// SIMATIC S7-200 SMART project (STEP 7-Micro/WIN SMART), CPU ST60

SYMBOL_TABLE 表格 1
RamZ             I0.0     // 压头零点
LeftStepPosLimit I0.1     // 左步进机构正限位
LeftStepNegaLimt I0.2     // 左步进机构负限位
RightStepPosLimit I0.3     // 右步进机构正限位
RightStepNegaLimt I0.4     // 右步进机构负限位
AirDownLimit     I0.5     // 气囊下限位
AirUpLimit       I0.6     // 气囊上限位
EMBotton         I0.7     // 急停
JOG1             I1.0     // JOG-
JOG2             I1.1     // JOG+
ResetBotton      I1.2     // 复位按钮
StartBotton      I1.3     // 循环启动
ManualBotton     I1.4     // 手动
AutoBotton       I1.5     // 自动
InderRunDone     I1.7     // 压头运行到位完成
Step1UpLimit     I2.0     // 步进机构气缸1上限位
Step1DownLimit   I2.1     // 步进机构气缸1下限位
Step2UpLimit     I2.2     // 步进机构气缸2上限位
Step2DownLimit   I2.3     // 步进机构气缸2下限位
LeftTopDownLimit I2.4     // 左顶尖气缸下限位
RightTopDownLimit I2.5     // 右顶尖气缸下限位
PipaBackLimit    I2.6     // 琵琶孔退回到位1
Ram1_Ready       I2.7     // 压头1伺服准备
Ram1_Alarm       I3.0     // 压头1驱动报警
Rot_Alarm        I3.1     // 旋转电机报警
Step_Alarm       I3.2     // 步进电机报警
PipaBackLimit2   I3.3     // 琵琶孔退回到位2
Ram2_Ready       I3.4     // 压头2伺服准备
Ram2_Alarm       I3.5     // 压头2驱动报警
Step_Send        I3.6     // 步进机构可送料信号
Step_First       I3.7     // 步进机构首端有料
Step_Middle      I4.0     // 校直机有料
Step_Last        I4.1     // 步进机构末端有料
LeftClamClose    I4.2     // 左夹爪气缸夹紧到位
RightClamClose   I4.3     // 右夹爪气缸夹紧到位
Press_Abnormal   I12.0    // 气压异常
FloatSup1BackLimit I12.1    // 浮动支撑1退回到位
FloatSup2BackLimit I12.2    // 浮动支撑2退回到位
FloatSup3BackLimit I12.3    // 浮动支撑3退回到位
FloatSup4BackLimit I12.4    // 浮动支撑4退回到位
FloatSup1FrontLimit I12.5    // 浮动支撑1前进到位
FloatSup2FrontLimit I12.6    // 浮动支撑2前进到位
FloatSup3FrontLimit I12.7    // 浮动支撑3前进到位
FloatSup4FrontLimit I16.0    // 浮动支撑4前进到位
YT5_BackLimit    I16.1    // 压头5缩回到位
YT4_BackLimit    I16.2    // 压头4缩回到位
YT3_BackLimit    I16.3    // 压头3缩回到位
YT2_BackLimit    I16.4    // 压头2缩回到位
YT1_BackLimit    I16.5    // 压头1缩回到位
LeftTopFloatLimit I16.6    // 左顶尖前进到位
LeftTopBackLimit I16.7    // 左顶尖退回到位
RightTopFloatLimit I17.0    // 右顶尖前进到位
RightTopBackLimit I17.1    // 右顶尖退回到位
找平到位             I17.3
步进后退             M11.0
步进前进             M11.2
主轴抬起             M11.4
主轴下压             M11.6
找平升              M12.0
支撑1进             M12.2
支撑2进             M12.3
支撑3进             M12.4
支撑4进             M12.5
一次抬起             M12.7
一次下压             M12.6
结束计时             M14.1
下压轴停止信号          M13.0
RamPULS          Q0.0     // 压头脉冲
StepPULS         Q0.1     // 左步进脉冲
RamSIGN          Q0.2     // 压头方向：高电位时压头下移，位移为正
RotaPULS         Q0.3     // 右步进电机脉冲
StartLamp        Q0.4     // 循环启动按钮灯
ServStart        Q0.5     // 启动
Ram_Rest         Q0.6     // 压头报警复位
Step_Sign        Q0.7     // 左步进机构方向
RotoSIGN         Q1.0     // 右旋转电机方向
YT1              Q1.2     // 1号压头气缸
YT2              Q1.3     // 2号压头气缸
YT3              Q1.4     // 3号压头气缸
YT4              Q1.5     // 4号压头气缸
YT5              Q1.6     // 5号压头气缸
Pipahole_Measure Q1.7     // 琵琶孔测量气缸
FloatSupport1    Q2.0     // 浮动支撑1缩回
FloatSupport2    Q2.1     // 浮动支撑2缩回
FloatSupport3    Q2.2     // 浮动支撑3缩回
FloatSupport4    Q2.3     // 浮动支撑4缩回
TopClamp         Q2.4     // 顶尖气缸夹紧
TopRelease       Q2.5     // 顶尖气缸松开
TopForward       Q2.6     // 顶尖气缸前进
Topback          Q2.7     // 顶尖气缸缩回
InderAirbagUp    Q8.0     // 压头气囊升起
InderAirbagDown  Q8.1     // 压头气囊落下
StepDown2        Q8.2     // 步进机构1落下
StepUp2          Q8.3     // 步进机构1升起
TopUp            Q8.4     // 顶尖气缸升起
TopDown          Q8.5     // 顶尖气缸落下
StepLast         Q8.6     // 步进机构末端可取料信号
FM               Q9.0     // 蜂鸣器
GREEN            Q9.1     // 绿灯
YELLOW           Q9.2     // 黄灯
RED              Q9.3     // 红灯
HG               Q9.4     // 加工合格
BHG              Q9.5     // 加工不合格
平升               Q12.0
左步进错误            VB300
右步进错误            VB304
下压轴错误            VB308
左步进速度            VD400
右步进速度            VD404
下压轴速度            VD408
左步进pos           VD412
右步进pos           VD416
下压轴pos           VD420
END_SYMBOL_TABLE

SYMBOL_TABLE 表格 2
HSC0_FREQ_PERIOD SMB196   // HSC0 频率测量周期: 0=1s 1=100ms 2=10ms
HSC0_TYPE        SMB195   // HSC0 类型: 0=计数 1=频率
HSC1_FREQ_PERIOD SMB198   // HSC1 频率测量周期: 0=1s 1=100ms 2=10ms
HSC1_TYPE        SMB197   // HSC1 类型: 0=计数 1=频率
HSC2_FREQ_PERIOD SMB200   // HSC2 频率测量周期: 0=1s 1=100ms 2=10ms
HSC2_TYPE        SMB199   // HSC2 类型: 0=计数 1=频率
HSC3_FREQ_PERIOD SMB202   // HSC3 频率测量周期: 0=1s 1=100ms 2=10ms
HSC3_TYPE        SMB201   // HSC3 类型: 0=计数 1=频率
HSC4_FREQ_PERIOD SMB204   // HSC4 频率测量周期: 0=1s 1=100ms 2=10ms
HSC4_TYPE        SMB203   // HSC4 类型: 0=计数 1=频率
HSC5_FREQ_PERIOD SMB206   // HSC5 频率测量周期: 0=1s 1=100ms 2=10ms
HSC5_TYPE        SMB205   // HSC5 类型: 0=计数 1=频率
PLS3_Abort_AE    SM580.4  // 由于添加错误终止 PTO2 包络：0 = 未终止；1 = 终止
PLS3_Ctrl        SMB581   // 监视和控制 Q0.2 的 PTO3（脉冲串输出）和 PWM3（脉冲宽度调制）
PLS3_Cycle       SMW582   // PWM3 周期值（2 到 65,535 个单位时基）；PTO3 频率值（1 到 65,535 Hz）
PLS3_Cycle_Update SM581.0  // PTO3/PWM3 更新周期或频率值：0 = 不更新；1 = 写入新周期/频率
PLS3_Disable_UC  SM580.5  // PTO3 用户在 PTO 包络运行过程中手动将其禁用 ：0 = 未禁用；1 = 手动禁用
PLS3_Enable      SM581.7  // PTO3/PWM3 使能：0 = 禁用；1 = 启用。
PLS3_Idle        SM580.7  // PTO3 空闲：0 = PTO 正在执行；1 = PTO 空闲。
PLS3_Ovr         SM580.6  // PTO3 管道上溢/下溢，管道为满时装载管道或传送空管道时：0 = 无溢出，1 = 管道上溢/下溢
PLS3_Select      SM581.6  // PTO3/PWM3 模式选择：0 = PWM；1 = PTO。
PTO3_Operation   SM581.5  // PTO3 选择单段/多段操作： 0 = 单段操作；1 = 多段操作
PTO3_PC          SMD586   // PTO3 脉冲计数值（1 到 2^32 - 1）
PTO3_PC_Update   SM581.2  // PTO3 更新脉冲计数值：0 = 不更新；1 = 写入新脉冲计数
PTO3_Profile_Offset SMW592   // PTO3 包络表的起始位置（从 V0 开始字节偏移）
PTO3_Seg_Num     SMB590   // 当前执行的 PTO3 包络的段数
PTO3_Status      SMB580   // PTO3 状态
PWM3_PW          SMW584   // PWM3 脉冲宽度值（0 到 65,535 个单位时基）
PWM3_PW_Update   SM581.1  // PWM3 更新脉冲宽度值：0 = 不更新；1 = 写入新脉冲宽度
PWM3_TimeBase    SM581.3  // PWM3 时基：0 = 1μs/刻度，1 = 1ms/刻度
END_SYMBOL_TABLE

SYMBOL_TABLE 表格 3
步进上料自锁           M0.0
夹正PC             M0.1
夹升PC             M0.2
夹反PC             M0.3
夹退PC             M0.4
夹停PC             M0.5
夹进PC             M0.6
夹紧PC             M0.7
夹降PC             M1.0
夹松PC             M1.1
步回零              M1.2
步最后PC            M1.3
步回零PC            M1.4
步最前PC            M1.5
步后PC             M1.6
步停PC             M1.7
步前PC             M2.0
步升PC             M2.1
步降PC             M2.2
axis0_dir        M2.3
压1进PC            M2.4
压1退PC            M2.5
压2进PC            M2.6
压2退PC            M2.7
压3进PC            M3.0
压3退PC            M3.1
压4进PC            M3.2
压4退PC            M3.3
压5进PC            M3.4
压5退PC            M3.5
压升PC             M3.6
压降PC             M3.7
压停PC             M4.0
压回零PC            M4.1
充气PC             M4.2
停充PC             M4.3
放气PC             M4.4
平升PC             M4.5
平停PC             M4.6
平降PC             M4.7
撑1进PC            M5.0
撑1停PC            M5.1
撑1退PC            M5.2
撑2进PC            M5.3
撑2停PC            M5.4
撑2退PC            M5.5
撑3进PC            M5.6
撑3停PC            M5.7
撑3退PC            M6.0
撑4进PC            M6.1
撑4停PC            M6.2
撑4退PC            M6.3
夹爪复位             M6.4
夹爪准备             M6.5
进出料              M6.6
压real            M6.7
有料未出             M7.0
机械INIT           M7.1
init_isrun       M7.2
axis1_dir        M7.3
axis0_动作         M7.4
axis1_动作         M7.5
急停               M7.6
压回零重设done        M7.7
左步进done          M8.0
右步进done          M8.1
下压轴done          M8.2
左步进dir           M8.3
右步进dir           M8.4
下压轴dir           M8.5
压回零done          M8.6
左步回零done         M8.7
右步回零done         M9.0
NG               M9.1
test             M9.2     // OK
OK               M9.3
找平ok             M9.4
备压PC             M9.5
传感器有料            M9.7
出料后有料            M10.0
下压isrun          M10.1
PLC_EN           M10.2
（先出）请求上料PC       M10.3
步进isrun          M10.4
夹爪isrun          M10.5
（不出）请求上料pc       M10.6
心跳               M30.0
下料信号             M30.1
下压量              MD20
END_SYMBOL_TABLE

SYMBOL_TABLE 表格 4
input1           V701.0
input2           V701.1
input3           V701.2
input4           V701.3
input5           V701.4
input6           V701.5
input7           V701.6
input8           V701.7
input9           V702.0
input10          V702.1
input11          V702.2
input12          V702.3
input13          V702.4
input14          V702.5
input15          V702.6
input16          V702.7
inputrel1        VD703
inputrel2        VD707
inputrel3        VD711
inputrel4        VD715
inputrel5        VD719
inputrel6        VD723
inputrel7        VD727
inputrel8        VD731
output1          V801.0
output2          V801.1
output3          V801.2
output4          V801.3
output5          V801.4
output6          V801.5
output7          V801.6
output8          V801.7
output9          V802.0
output10         V802.1
output11         V802.2
output12         V802.3
output13         V802.4
output14         V802.5
output15         V802.6
output16         V802.7
outputrel1       VD803
outputrel2       VD807
outputrel3       VD811
outputrel4       VD815
outputrel5       VD819
outputrel6       VD823
outputrel7       VD827
outputrel8       VD831
END_SYMBOL_TABLE

ORGANIZATION_BLOCK MAIN:OB1
TITLE=程序注释
BEGIN
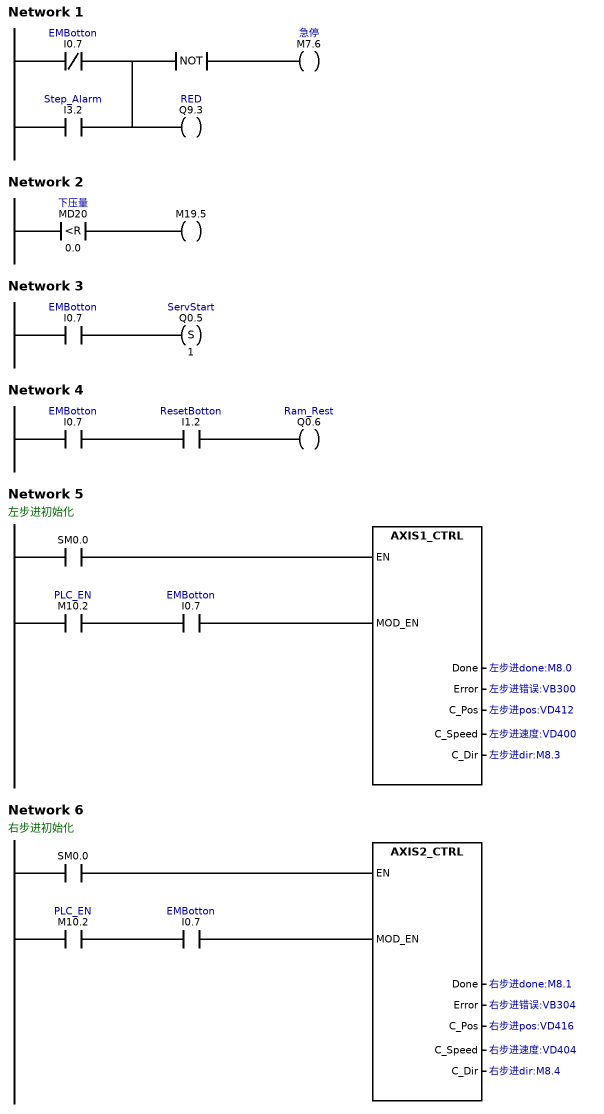
Network 1
LDN    EMBotton:I0.7
O      Step_Alarm:I3.2
LPS
NOT
=      急停:M7.6
LPP
=      RED:Q9.3
Network 2
LDR<   下压量:MD20, 0.0
=      M19.5
Network 3
LD     EMBotton:I0.7
S      ServStart:Q0.5, 1
Network 4
LD     EMBotton:I0.7
A      ResetBotton:I1.2
=      Ram_Rest:Q0.6
Network 5
// 左步进初始化
LD     SM0.0
=      L60.0
LD     PLC_EN:M10.2
A      EMBotton:I0.7
=      L63.7
LD     L60.0
CALL   AXIS1_CTRL:SBR12, L63.7, 左步进done:M8.0, 左步进错误:VB300, 左步进pos:VD412, 左步进速度:VD400, 左步进dir:M8.3
Network 6
// 右步进初始化
LD     SM0.0
=      L60.0
LD     PLC_EN:M10.2
A      EMBotton:I0.7
=      L63.7
LD     L60.0
CALL   AXIS2_CTRL:SBR23, L63.7, 右步进done:M8.1, 右步进错误:VB304, 右步进pos:VD416, 右步进速度:VD404, 右步进dir:M8.4
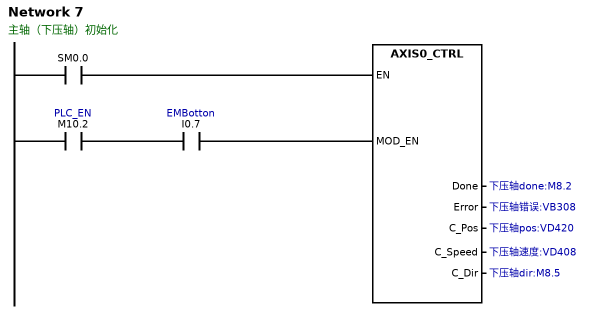
Network 7
// 主轴（下压轴）初始化
LD     SM0.0
=      L60.0
LD     PLC_EN:M10.2
A      EMBotton:I0.7
=      L63.7
LD     L60.0
CALL   AXIS0_CTRL:SBR4, L63.7, 下压轴done:M8.2, 下压轴错误:VB308, 下压轴pos:VD420, 下压轴速度:VD408, 下压轴dir:M8.5
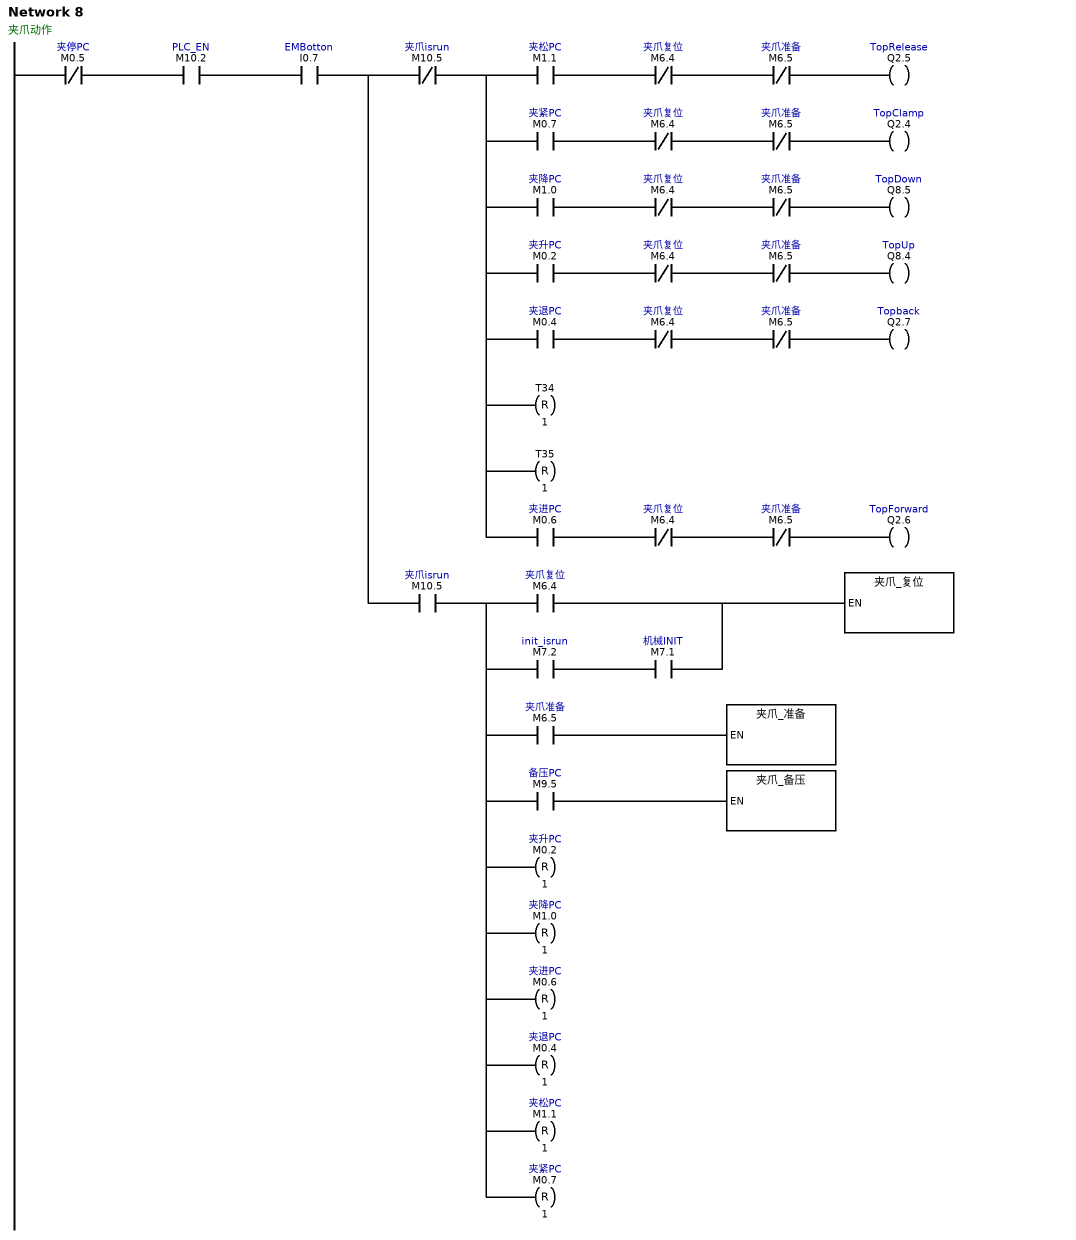
Network 8
// 夹爪动作
LDN    夹停PC:M0.5
A      PLC_EN:M10.2
A      EMBotton:I0.7
LPS
AN     夹爪isrun:M10.5
LPS
A      夹松PC:M1.1
AN     夹爪复位:M6.4
AN     夹爪准备:M6.5
=      TopRelease:Q2.5
LRD
A      夹紧PC:M0.7
AN     夹爪复位:M6.4
AN     夹爪准备:M6.5
=      TopClamp:Q2.4
LRD
A      夹降PC:M1.0
AN     夹爪复位:M6.4
AN     夹爪准备:M6.5
=      TopDown:Q8.5
LRD
A      夹升PC:M0.2
AN     夹爪复位:M6.4
AN     夹爪准备:M6.5
=      TopUp:Q8.4
LRD
A      夹退PC:M0.4
AN     夹爪复位:M6.4
AN     夹爪准备:M6.5
=      Topback:Q2.7
LRD
R      T34, 1
LRD
R      T35, 1
LPP
A      夹进PC:M0.6
AN     夹爪复位:M6.4
AN     夹爪准备:M6.5
=      TopForward:Q2.6
LPP
A      夹爪isrun:M10.5
LPS
LD     夹爪复位:M6.4
LD     init_isrun:M7.2
A      机械INIT:M7.1
OLD
ALD
CALL   夹爪_复位:SBR0
LPP
LPS
A      夹爪准备:M6.5
CALL   夹爪_准备:SBR1
LRD
A      备压PC:M9.5
CALL   夹爪_备压:SBR35
LRD
R      夹升PC:M0.2, 1
LRD
R      夹降PC:M1.0, 1
LRD
R      夹进PC:M0.6, 1
LRD
R      夹退PC:M0.4, 1
LRD
R      夹松PC:M1.1, 1
LPP
R      夹紧PC:M0.7, 1
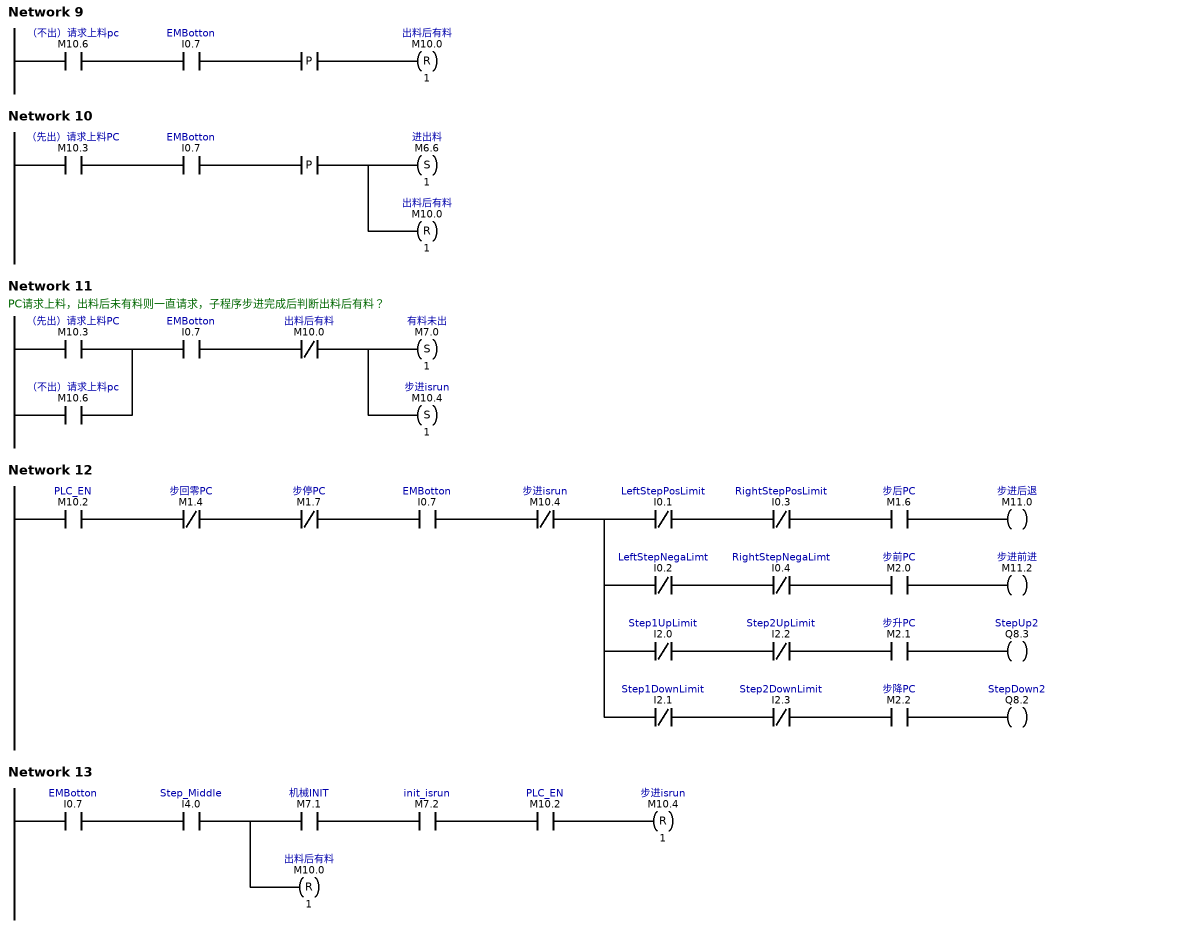
Network 9
LD     （不出）请求上料pc:M10.6
A      EMBotton:I0.7
EU
R      出料后有料:M10.0, 1
Network 10
LD     （先出）请求上料PC:M10.3
A      EMBotton:I0.7
EU
S      进出料:M6.6, 1
R      出料后有料:M10.0, 1
Network 11
// PC请求上料，出料后未有料则一直请求，子程序步进完成后判断出料后有料？
LD     （先出）请求上料PC:M10.3
O      （不出）请求上料pc:M10.6
A      EMBotton:I0.7
AN     出料后有料:M10.0
S      有料未出:M7.0, 1
S      步进isrun:M10.4, 1
Network 12
LD     PLC_EN:M10.2
AN     步回零PC:M1.4
AN     步停PC:M1.7
A      EMBotton:I0.7
AN     步进isrun:M10.4
LPS
AN     LeftStepPosLimit:I0.1
AN     RightStepPosLimit:I0.3
A      步后PC:M1.6
=      步进后退:M11.0
LRD
AN     LeftStepNegaLimt:I0.2
AN     RightStepNegaLimt:I0.4
A      步前PC:M2.0
=      步进前进:M11.2
LRD
AN     Step1UpLimit:I2.0
AN     Step2UpLimit:I2.2
A      步升PC:M2.1
=      StepUp2:Q8.3
LPP
AN     Step1DownLimit:I2.1
AN     Step2DownLimit:I2.3
A      步降PC:M2.2
=      StepDown2:Q8.2
Network 13
LD     EMBotton:I0.7
A      Step_Middle:I4.0
LPS
A      机械INIT:M7.1
A      init_isrun:M7.2
A      PLC_EN:M10.2
R      步进isrun:M10.4, 1
LPP
R      出料后有料:M10.0, 1
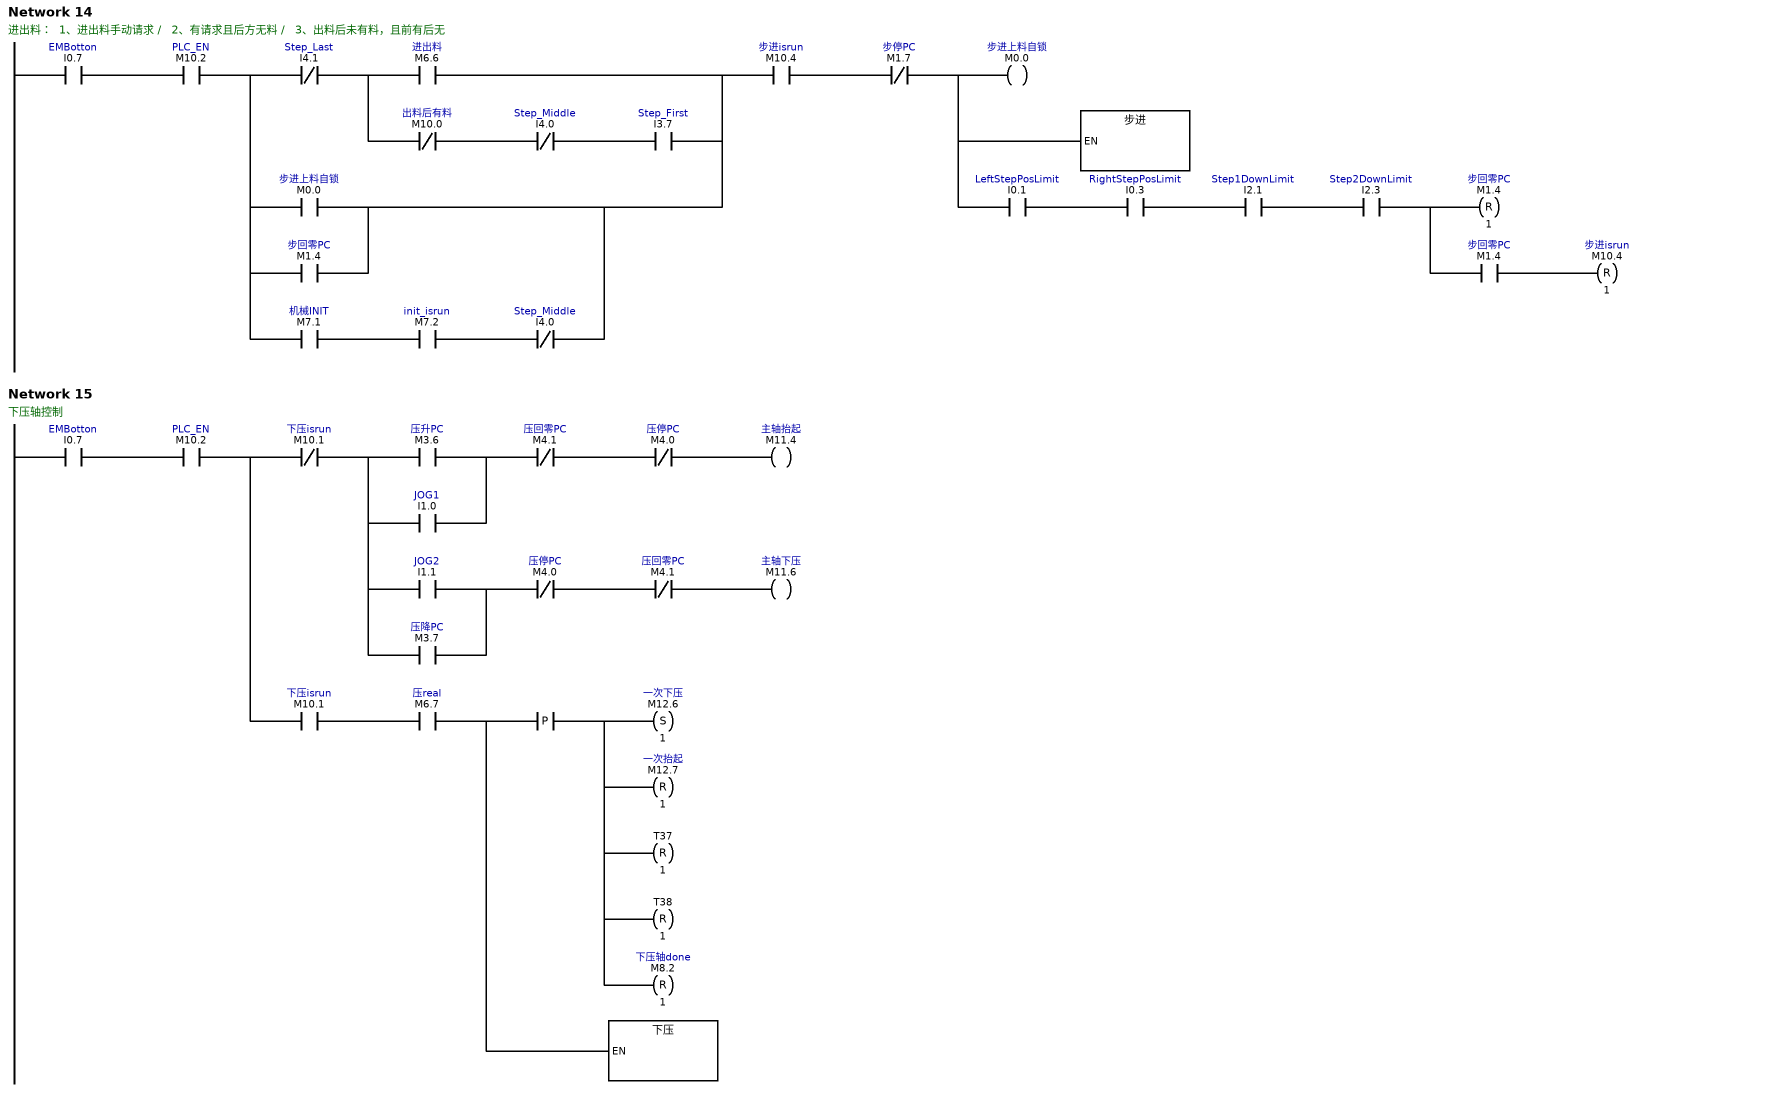
Network 14
// 进出料：	1、进出料手动请求
// 	2、有请求且后方无料
// 	3、出料后未有料，且前有后无
LD     EMBotton:I0.7
A      PLC_EN:M10.2
LDN    Step_Last:I4.1
LD     进出料:M6.6
LDN    出料后有料:M10.0
AN     Step_Middle:I4.0
A      Step_First:I3.7
OLD
ALD
LD     步进上料自锁:M0.0
O      步回零PC:M1.4
LD     机械INIT:M7.1
A      init_isrun:M7.2
AN     Step_Middle:I4.0
OLD
OLD
ALD
A      步进isrun:M10.4
AN     步停PC:M1.7
=      步进上料自锁:M0.0
CALL   步进:SBR2
A      LeftStepPosLimit:I0.1
A      RightStepPosLimit:I0.3
A      Step1DownLimit:I2.1
A      Step2DownLimit:I2.3
R      步回零PC:M1.4, 1
A      步回零PC:M1.4
R      步进isrun:M10.4, 1
Network 15
// 下压轴控制
LD     EMBotton:I0.7
A      PLC_EN:M10.2
LPS
AN     下压isrun:M10.1
LPS
LD     压升PC:M3.6
O      JOG1:I1.0
ALD
AN     压回零PC:M4.1
AN     压停PC:M4.0
=      主轴抬起:M11.4
LPP
LD     JOG2:I1.1
O      压降PC:M3.7
ALD
AN     压停PC:M4.0
AN     压回零PC:M4.1
=      主轴下压:M11.6
LPP
A      下压isrun:M10.1
A      压real:M6.7
LPS
EU
S      一次下压:M12.6, 1
R      一次抬起:M12.7, 1
R      T37, 1
R      T38, 1
R      下压轴done:M8.2, 1
LPP
CALL   下压:SBR3
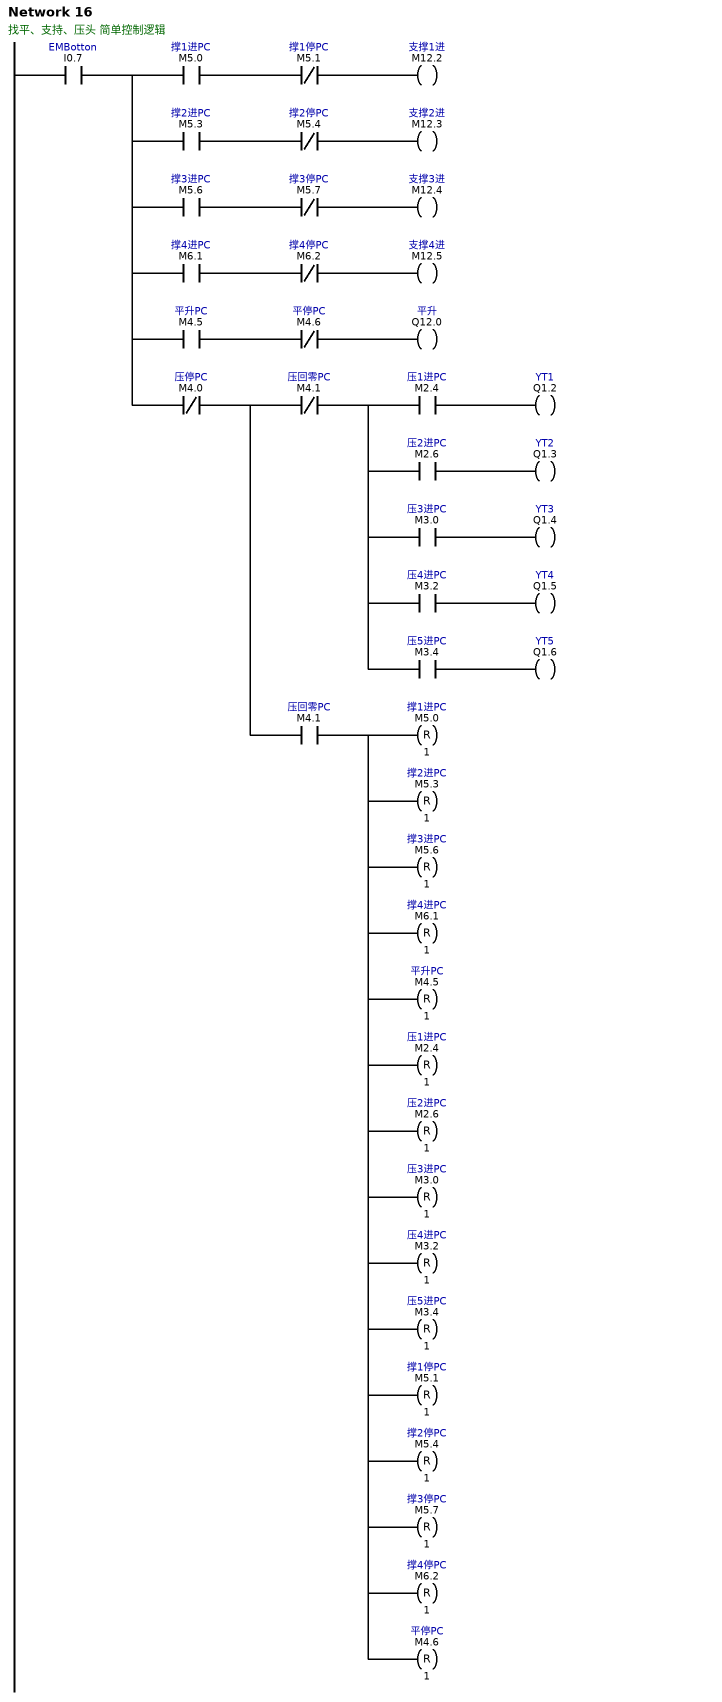
Network 16
// 找平、支持、压头 简单控制逻辑
LD     EMBotton:I0.7
LPS
A      撑1进PC:M5.0
AN     撑1停PC:M5.1
=      支撑1进:M12.2
LRD
A      撑2进PC:M5.3
AN     撑2停PC:M5.4
=      支撑2进:M12.3
LRD
A      撑3进PC:M5.6
AN     撑3停PC:M5.7
=      支撑3进:M12.4
LRD
A      撑4进PC:M6.1
AN     撑4停PC:M6.2
=      支撑4进:M12.5
LRD
A      平升PC:M4.5
AN     平停PC:M4.6
=      平升:Q12.0
LPP
AN     压停PC:M4.0
LPS
AN     压回零PC:M4.1
LPS
A      压1进PC:M2.4
=      YT1:Q1.2
LRD
A      压2进PC:M2.6
=      YT2:Q1.3
LRD
A      压3进PC:M3.0
=      YT3:Q1.4
LRD
A      压4进PC:M3.2
=      YT4:Q1.5
LPP
A      压5进PC:M3.4
=      YT5:Q1.6
LPP
A      压回零PC:M4.1
R      撑1进PC:M5.0, 1
R      撑2进PC:M5.3, 1
R      撑3进PC:M5.6, 1
R      撑4进PC:M6.1, 1
R      平升PC:M4.5, 1
R      压1进PC:M2.4, 1
R      压2进PC:M2.6, 1
R      压3进PC:M3.0, 1
R      压4进PC:M3.2, 1
R      压5进PC:M3.4, 1
R      撑1停PC:M5.1, 1
R      撑2停PC:M5.4, 1
R      撑3停PC:M5.7, 1
R      撑4停PC:M6.2, 1
R      平停PC:M4.6, 1
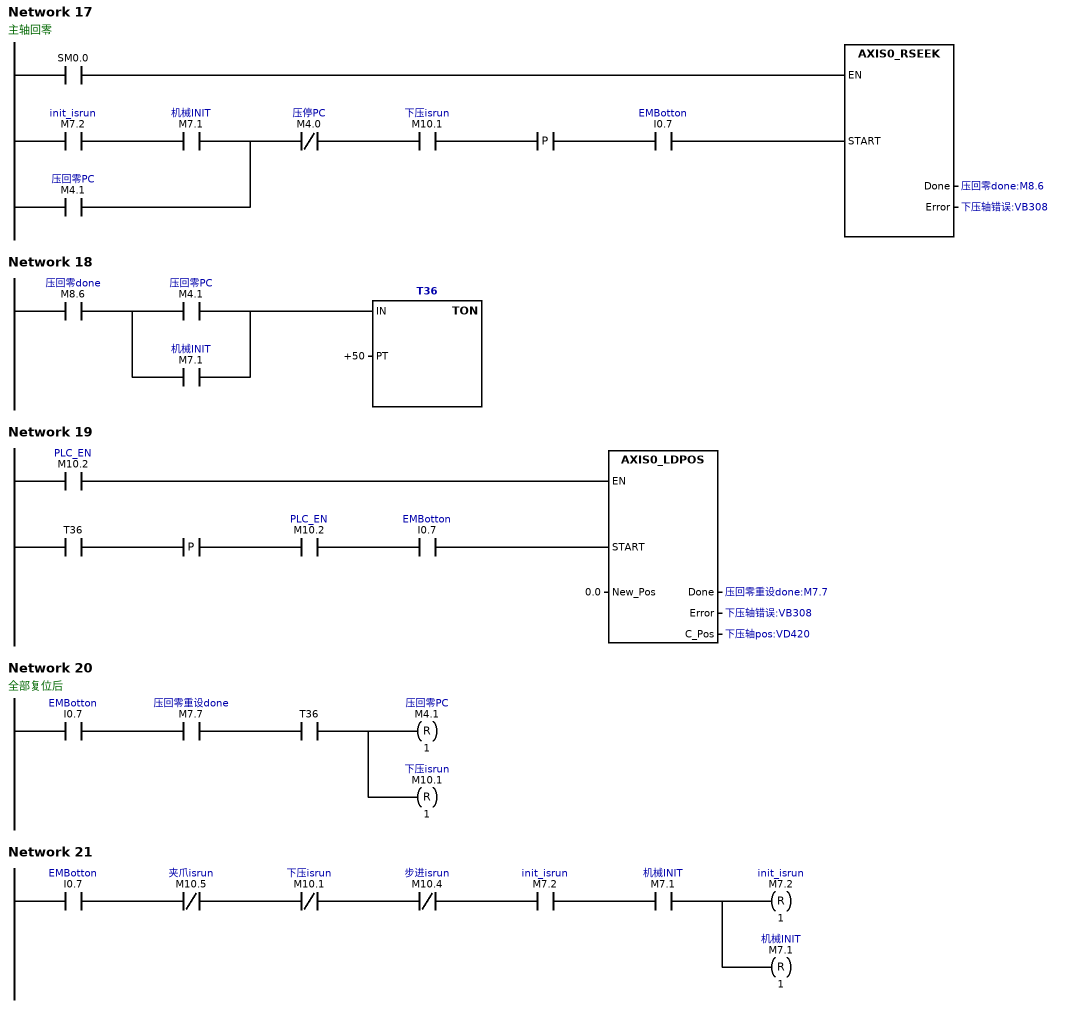
Network 17
// 主轴回零
LD     SM0.0
=      L60.0
LD     init_isrun:M7.2
A      机械INIT:M7.1
O      压回零PC:M4.1
AN     压停PC:M4.0
A      下压isrun:M10.1
EU
A      EMBotton:I0.7
=      L63.7
LD     L60.0
CALL   AXIS0_RSEEK:SBR7, L63.7, 压回零done:M8.6, 下压轴错误:VB308
Network 18
LD     压回零done:M8.6
LD     压回零PC:M4.1
O      机械INIT:M7.1
ALD
TON    T36, +50
Network 19
LD     PLC_EN:M10.2
=      L60.0
LD     T36
EU
A      PLC_EN:M10.2
A      EMBotton:I0.7
=      L63.7
LD     L60.0
CALL   AXIS0_LDPOS:SBR9, L63.7, 0.0, 压回零重设done:M7.7, 下压轴错误:VB308, 下压轴pos:VD420
Network 20
// 全部复位后
LD     EMBotton:I0.7
A      压回零重设done:M7.7
A      T36
R      压回零PC:M4.1, 1
R      下压isrun:M10.1, 1
Network 21
LD     EMBotton:I0.7
AN     夹爪isrun:M10.5
AN     下压isrun:M10.1
AN     步进isrun:M10.4
A      init_isrun:M7.2
A      机械INIT:M7.1
R      init_isrun:M7.2, 1
R      机械INIT:M7.1, 1
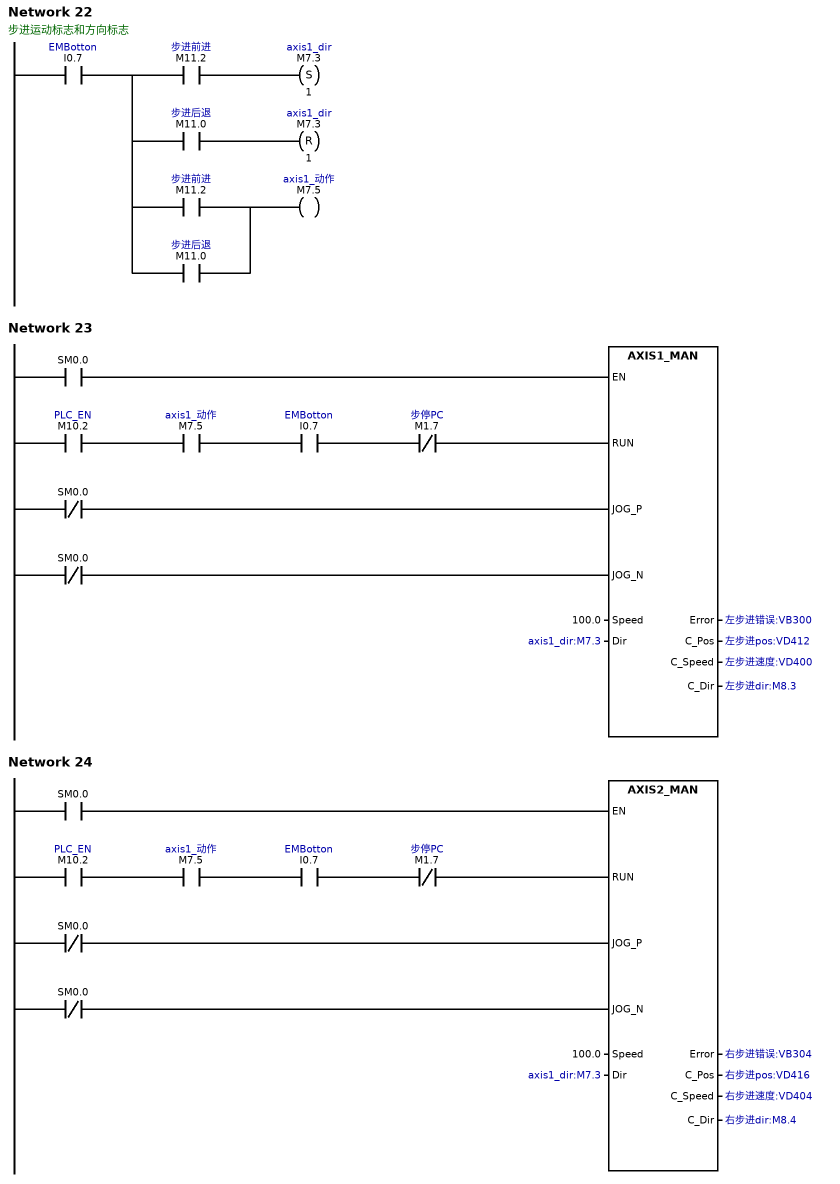
Network 22
// 步进运动标志和方向标志
LD     EMBotton:I0.7
LPS
A      步进前进:M11.2
S      axis1_dir:M7.3, 1
LRD
A      步进后退:M11.0
R      axis1_dir:M7.3, 1
LPP
LD     步进前进:M11.2
O      步进后退:M11.0
ALD
=      axis1_动作:M7.5
Network 23
LD     SM0.0
=      L60.0
LD     PLC_EN:M10.2
A      axis1_动作:M7.5
A      EMBotton:I0.7
AN     步停PC:M1.7
=      L63.7
LDN    SM0.0
=      L63.6
LDN    SM0.0
=      L63.5
LD     L60.0
CALL   AXIS1_MAN:SBR13, L63.7, L63.6, L63.5, 100.0, axis1_dir:M7.3, 左步进错误:VB300, 左步进pos:VD412, 左步进速度:VD400, 左步进dir:M8.3
Network 24
LD     SM0.0
=      L60.0
LD     PLC_EN:M10.2
A      axis1_动作:M7.5
A      EMBotton:I0.7
AN     步停PC:M1.7
=      L63.7
LDN    SM0.0
=      L63.6
LDN    SM0.0
=      L63.5
LD     L60.0
CALL   AXIS2_MAN:SBR24, L63.7, L63.6, L63.5, 100.0, axis1_dir:M7.3, 右步进错误:VB304, 右步进pos:VD416, 右步进速度:VD404, 右步进dir:M8.4
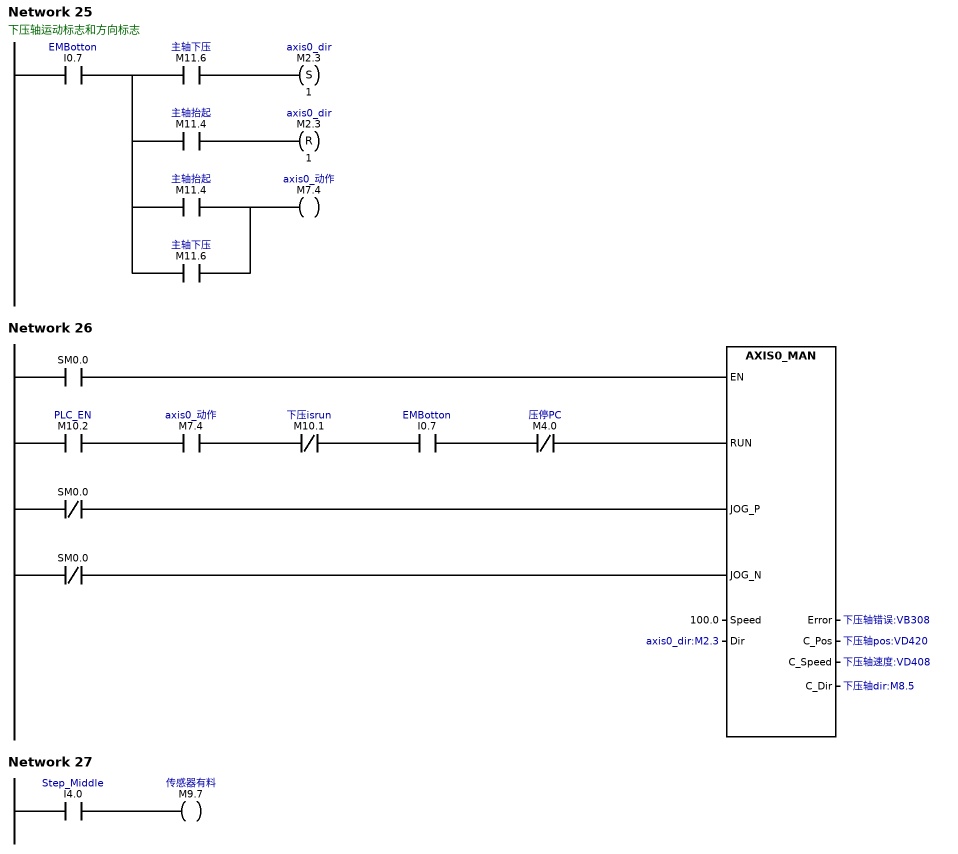
Network 25
// 下压轴运动标志和方向标志
LD     EMBotton:I0.7
LPS
A      主轴下压:M11.6
S      axis0_dir:M2.3, 1
LRD
A      主轴抬起:M11.4
R      axis0_dir:M2.3, 1
LPP
LD     主轴抬起:M11.4
O      主轴下压:M11.6
ALD
=      axis0_动作:M7.4
Network 26
LD     SM0.0
=      L60.0
LD     PLC_EN:M10.2
A      axis0_动作:M7.4
AN     下压isrun:M10.1
A      EMBotton:I0.7
AN     压停PC:M4.0
=      L63.7
LDN    SM0.0
=      L63.6
LDN    SM0.0
=      L63.5
LD     L60.0
CALL   AXIS0_MAN:SBR5, L63.7, L63.6, L63.5, 100.0, axis0_dir:M2.3, 下压轴错误:VB308, 下压轴pos:VD420, 下压轴速度:VD408, 下压轴dir:M8.5
Network 27
LD     Step_Middle:I4.0
=      传感器有料:M9.7
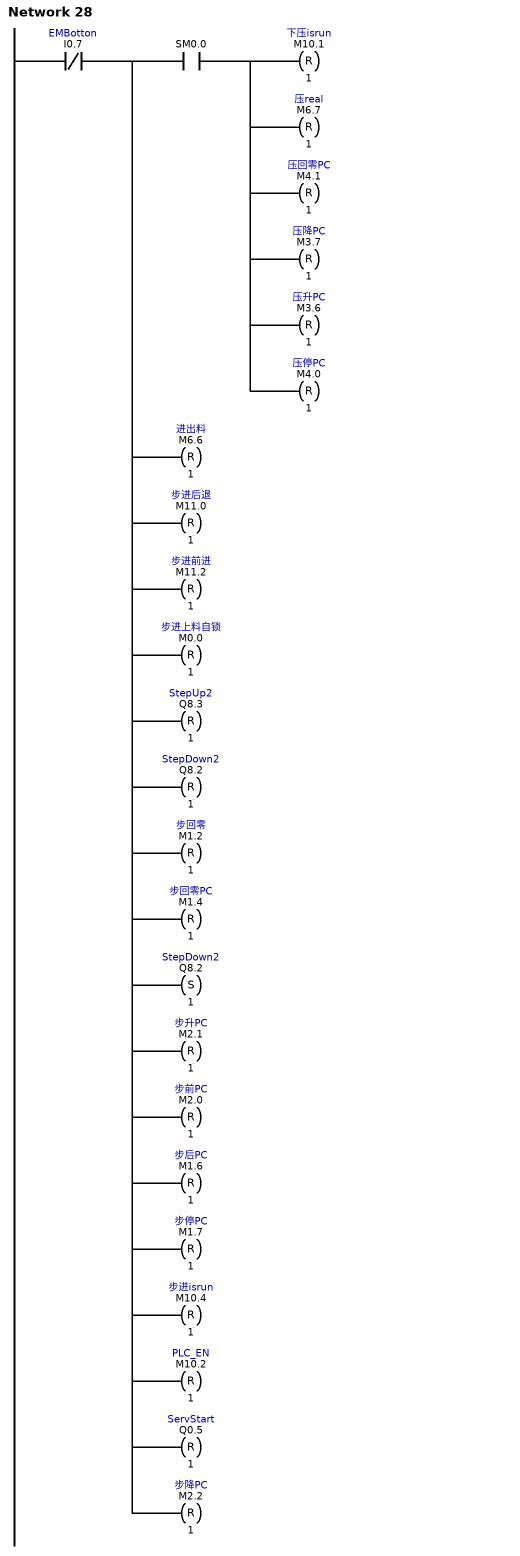
Network 28
LDN    EMBotton:I0.7
LPS
A      SM0.0
R      下压isrun:M10.1, 1
R      压real:M6.7, 1
R      压回零PC:M4.1, 1
R      压降PC:M3.7, 1
R      压升PC:M3.6, 1
R      压停PC:M4.0, 1
LPP
R      进出料:M6.6, 1
R      步进后退:M11.0, 1
R      步进前进:M11.2, 1
R      步进上料自锁:M0.0, 1
R      StepUp2:Q8.3, 1
R      StepDown2:Q8.2, 1
R      步回零:M1.2, 1
R      步回零PC:M1.4, 1
S      StepDown2:Q8.2, 1
R      步升PC:M2.1, 1
R      步前PC:M2.0, 1
R      步后PC:M1.6, 1
R      步停PC:M1.7, 1
R      步进isrun:M10.4, 1
R      PLC_EN:M10.2, 1
R      ServStart:Q0.5, 1
R      步降PC:M2.2, 1
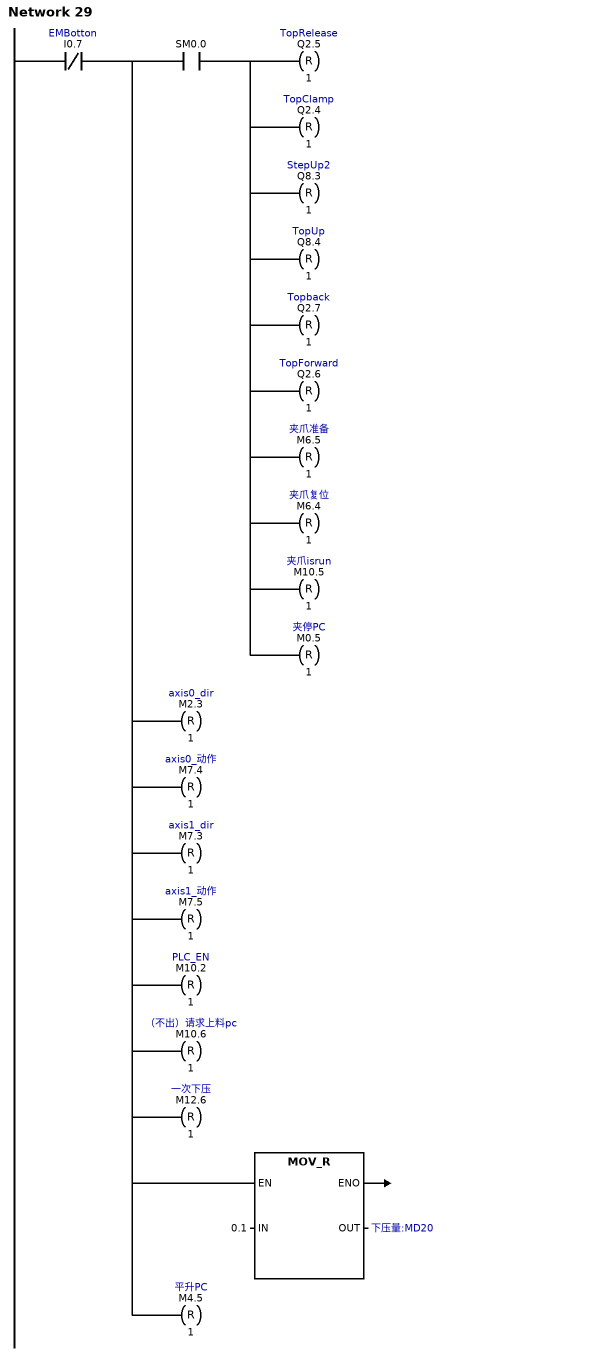
Network 29
LDN    EMBotton:I0.7
LPS
A      SM0.0
R      TopRelease:Q2.5, 1
R      TopClamp:Q2.4, 1
R      StepUp2:Q8.3, 1
R      TopUp:Q8.4, 1
R      Topback:Q2.7, 1
R      TopForward:Q2.6, 1
R      夹爪准备:M6.5, 1
R      夹爪复位:M6.4, 1
R      夹爪isrun:M10.5, 1
R      夹停PC:M0.5, 1
LPP
R      axis0_dir:M2.3, 1
R      axis0_动作:M7.4, 1
R      axis1_dir:M7.3, 1
R      axis1_动作:M7.5, 1
R      PLC_EN:M10.2, 1
R      （不出）请求上料pc:M10.6, 1
R      一次下压:M12.6, 1
MOVR   0.1, 下压量:MD20
R      平升PC:M4.5, 1
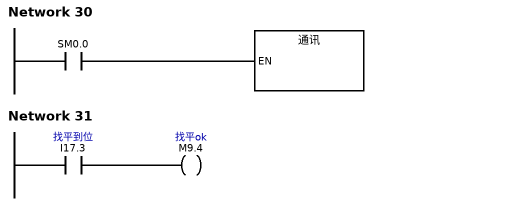
Network 30
LD     SM0.0
CALL   通讯:SBR34
Network 31
LD     找平到位:I17.3
=      找平ok:M9.4
END_ORGANIZATION_BLOCK

SUBROUTINE_BLOCK 夹爪_复位:SBR0
TITLE=单检一周复位
BEGIN
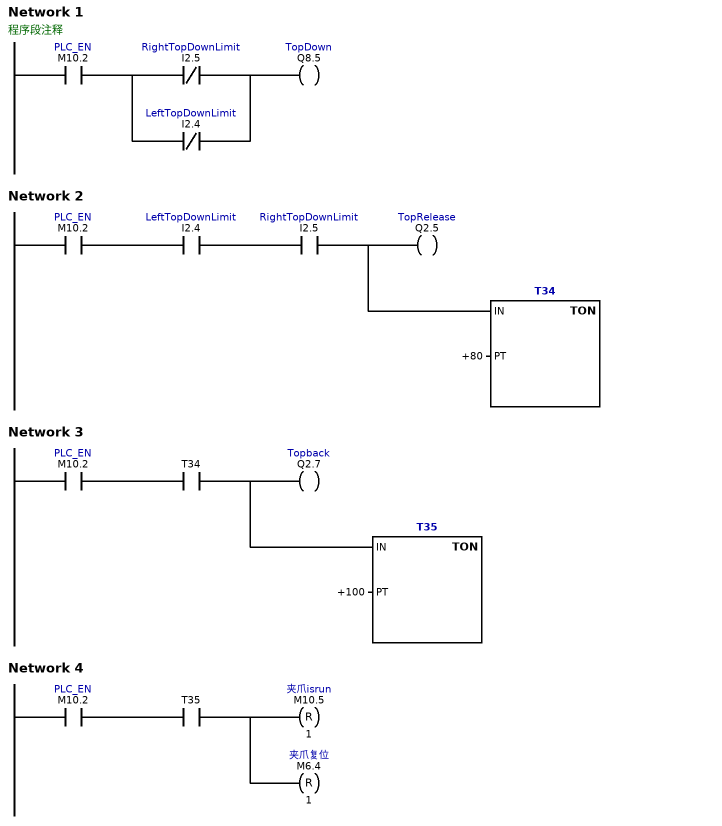
Network 1
// 程序段注释
LD     PLC_EN:M10.2
LDN    RightTopDownLimit:I2.5
ON     LeftTopDownLimit:I2.4
ALD
=      TopDown:Q8.5
Network 2
LD     PLC_EN:M10.2
A      LeftTopDownLimit:I2.4
A      RightTopDownLimit:I2.5
=      TopRelease:Q2.5
TON    T34, +80
Network 3
LD     PLC_EN:M10.2
A      T34
=      Topback:Q2.7
TON    T35, +100
Network 4
LD     PLC_EN:M10.2
A      T35
R      夹爪isrun:M10.5, 1
R      夹爪复位:M6.4, 1
END_SUBROUTINE_BLOCK

SUBROUTINE_BLOCK 夹爪_准备:SBR1
TITLE=单检一周准备
BEGIN
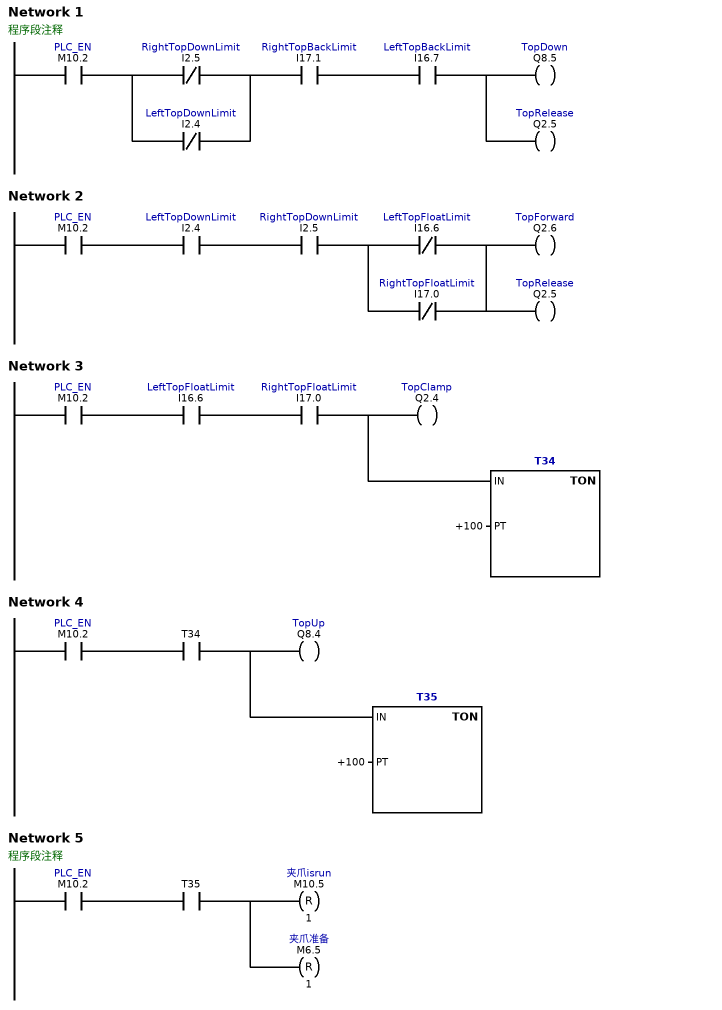
Network 1
// 程序段注释
LD     PLC_EN:M10.2
LDN    RightTopDownLimit:I2.5
ON     LeftTopDownLimit:I2.4
ALD
A      RightTopBackLimit:I17.1
A      LeftTopBackLimit:I16.7
=      TopDown:Q8.5
=      TopRelease:Q2.5
Network 2
LD     PLC_EN:M10.2
A      LeftTopDownLimit:I2.4
A      RightTopDownLimit:I2.5
LDN    LeftTopFloatLimit:I16.6
ON     RightTopFloatLimit:I17.0
ALD
=      TopForward:Q2.6
=      TopRelease:Q2.5
Network 3
LD     PLC_EN:M10.2
A      LeftTopFloatLimit:I16.6
A      RightTopFloatLimit:I17.0
=      TopClamp:Q2.4
TON    T34, +100
Network 4
LD     PLC_EN:M10.2
A      T34
=      TopUp:Q8.4
TON    T35, +100
Network 5
// 程序段注释
LD     PLC_EN:M10.2
A      T35
R      夹爪isrun:M10.5, 1
R      夹爪准备:M6.5, 1
END_SUBROUTINE_BLOCK

SUBROUTINE_BLOCK 步进:SBR2
TITLE=进料/出料
BEGIN
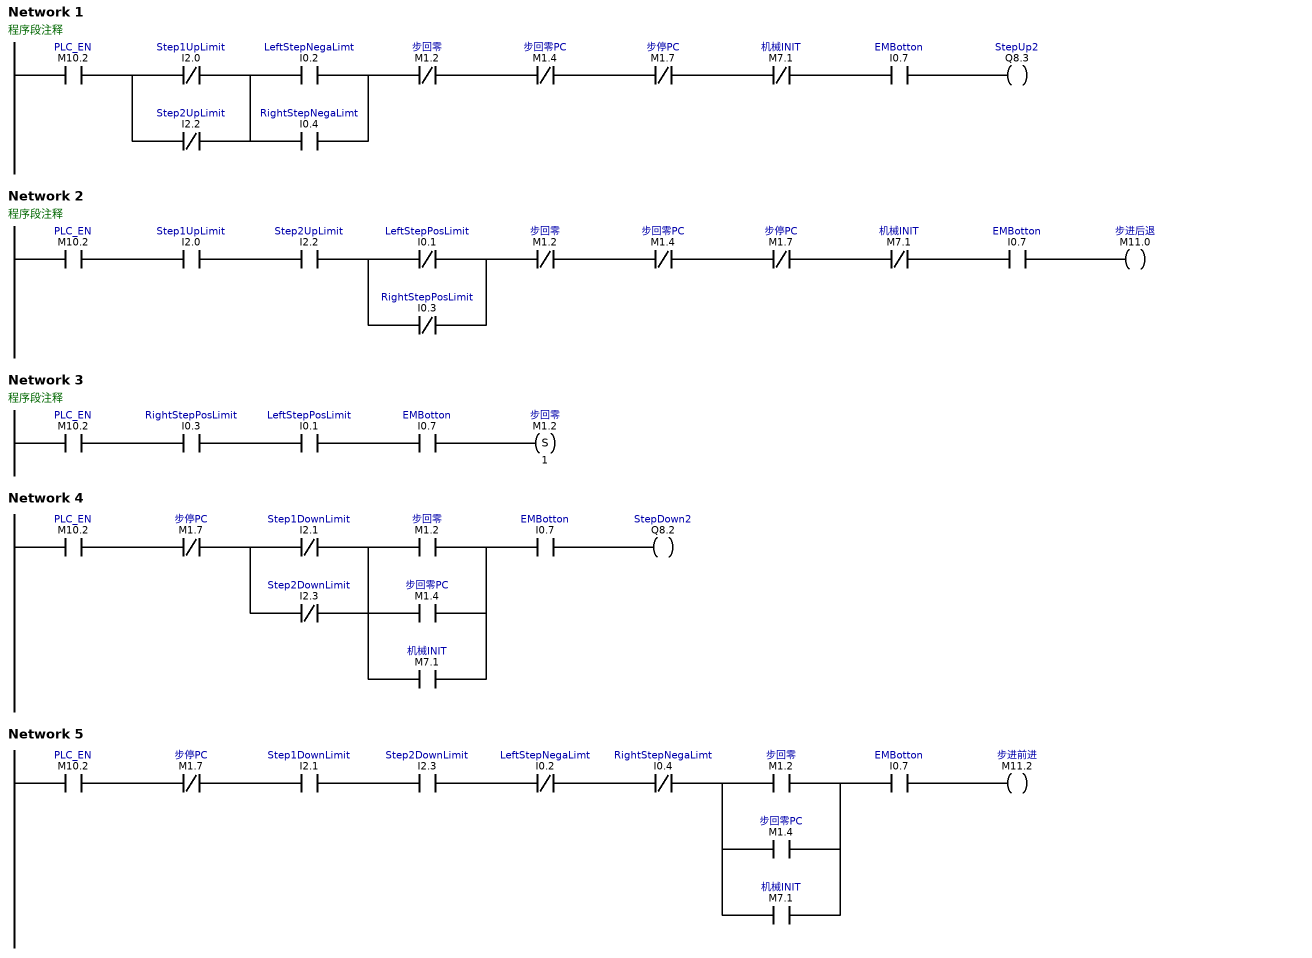
Network 1
// 程序段注释
LD     PLC_EN:M10.2
LDN    Step1UpLimit:I2.0
ON     Step2UpLimit:I2.2
ALD
LD     LeftStepNegaLimt:I0.2
O      RightStepNegaLimt:I0.4
ALD
AN     步回零:M1.2
AN     步回零PC:M1.4
AN     步停PC:M1.7
AN     机械INIT:M7.1
A      EMBotton:I0.7
=      StepUp2:Q8.3
Network 2
// 程序段注释
LD     PLC_EN:M10.2
A      Step1UpLimit:I2.0
A      Step2UpLimit:I2.2
LDN    LeftStepPosLimit:I0.1
ON     RightStepPosLimit:I0.3
ALD
AN     步回零:M1.2
AN     步回零PC:M1.4
AN     步停PC:M1.7
AN     机械INIT:M7.1
A      EMBotton:I0.7
=      步进后退:M11.0
Network 3
// 程序段注释
LD     PLC_EN:M10.2
A      RightStepPosLimit:I0.3
A      LeftStepPosLimit:I0.1
A      EMBotton:I0.7
S      步回零:M1.2, 1
Network 4
LD     PLC_EN:M10.2
AN     步停PC:M1.7
LDN    Step1DownLimit:I2.1
ON     Step2DownLimit:I2.3
ALD
LD     步回零:M1.2
O      步回零PC:M1.4
O      机械INIT:M7.1
ALD
A      EMBotton:I0.7
=      StepDown2:Q8.2
Network 5
LD     PLC_EN:M10.2
AN     步停PC:M1.7
A      Step1DownLimit:I2.1
A      Step2DownLimit:I2.3
AN     LeftStepNegaLimt:I0.2
AN     RightStepNegaLimt:I0.4
LD     步回零:M1.2
O      步回零PC:M1.4
O      机械INIT:M7.1
ALD
A      EMBotton:I0.7
=      步进前进:M11.2
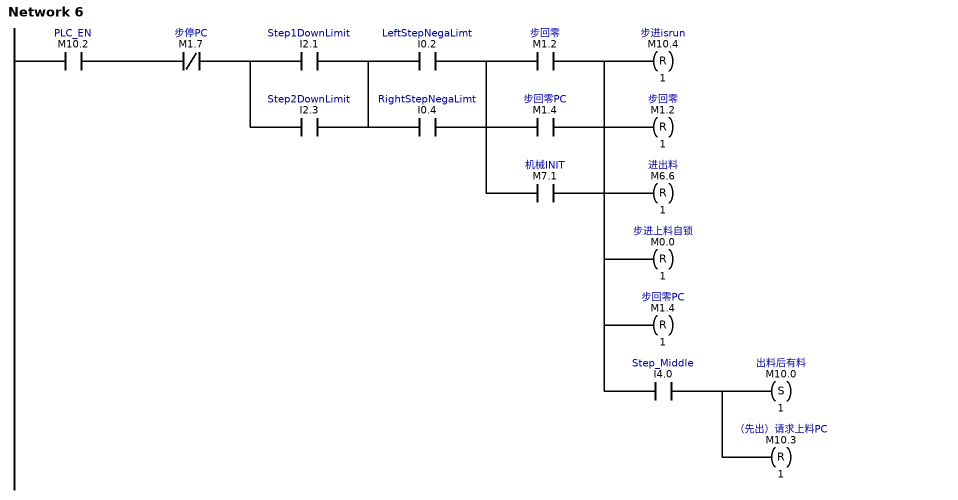
Network 6
LD     PLC_EN:M10.2
AN     步停PC:M1.7
LD     Step1DownLimit:I2.1
O      Step2DownLimit:I2.3
ALD
LD     LeftStepNegaLimt:I0.2
O      RightStepNegaLimt:I0.4
ALD
LD     步回零:M1.2
O      步回零PC:M1.4
O      机械INIT:M7.1
ALD
R      步进isrun:M10.4, 1
R      步回零:M1.2, 1
R      进出料:M6.6, 1
R      步进上料自锁:M0.0, 1
R      步回零PC:M1.4, 1
A      Step_Middle:I4.0
S      出料后有料:M10.0, 1
R      （先出）请求上料PC:M10.3, 1
END_SUBROUTINE_BLOCK

SUBROUTINE_BLOCK 下压:SBR3
TITLE=下压动作
BEGIN
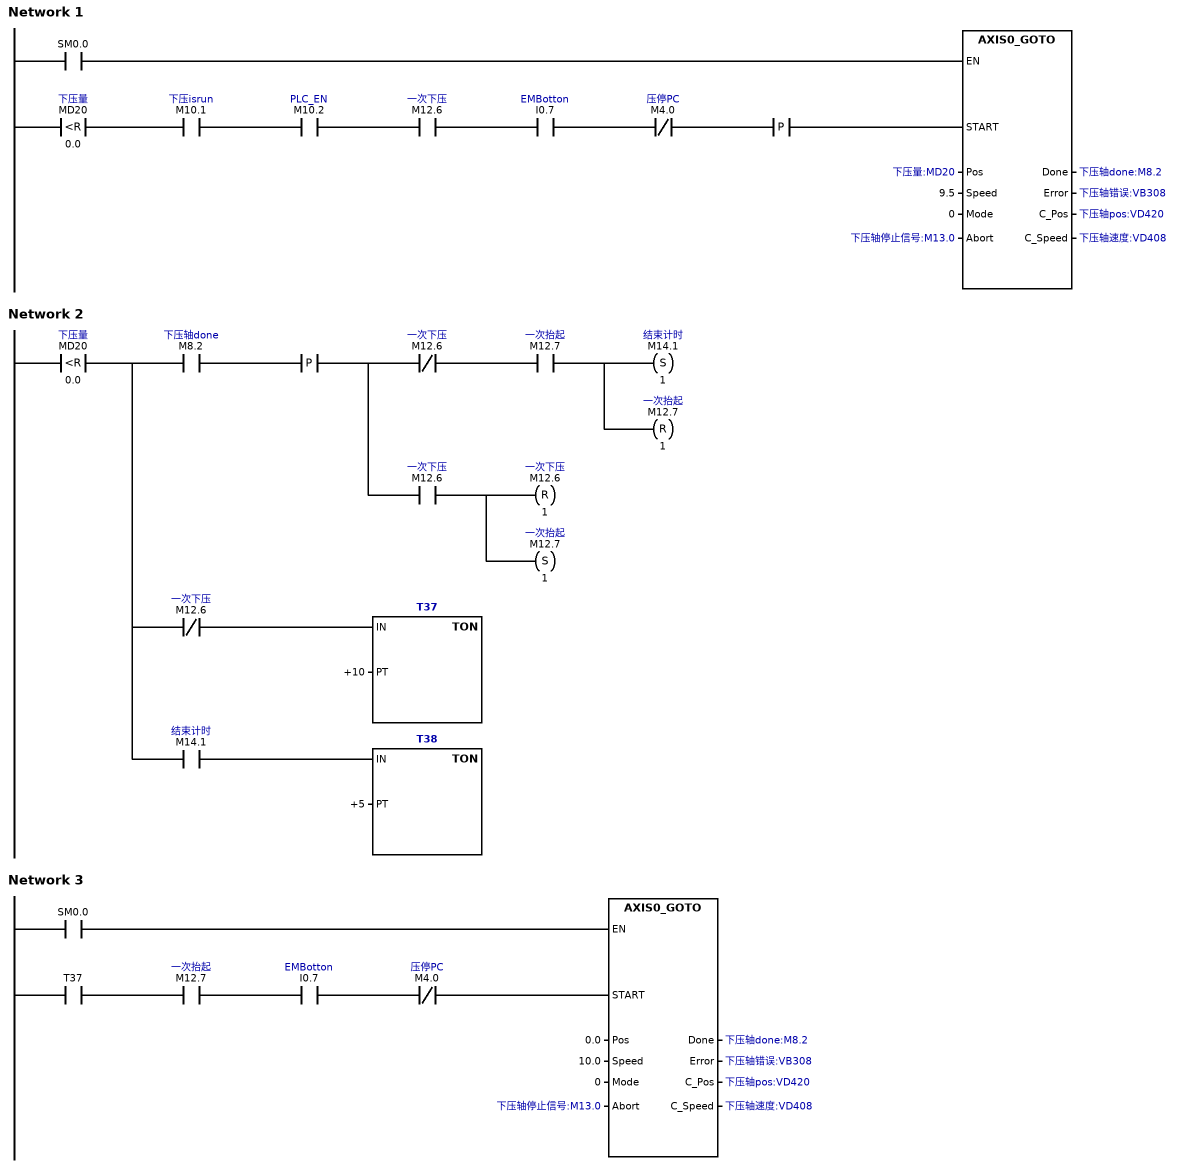
Network 1
LD     SM0.0
=      L60.0
LDR<   下压量:MD20, 0.0
A      下压isrun:M10.1
A      PLC_EN:M10.2
A      一次下压:M12.6
A      EMBotton:I0.7
AN     压停PC:M4.0
EU
=      L63.7
LD     L60.0
CALL   AXIS0_GOTO:SBR6, L63.7, 下压量:MD20, 9.5, 0, 下压轴停止信号:M13.0, 下压轴done:M8.2, 下压轴错误:VB308, 下压轴pos:VD420, 下压轴速度:VD408
Network 2
LDR<   下压量:MD20, 0.0
LPS
A      下压轴done:M8.2
EU
LPS
AN     一次下压:M12.6
A      一次抬起:M12.7
S      结束计时:M14.1, 1
R      一次抬起:M12.7, 1
LPP
A      一次下压:M12.6
R      一次下压:M12.6, 1
S      一次抬起:M12.7, 1
LPP
LPS
AN     一次下压:M12.6
TON    T37, +10
LPP
A      结束计时:M14.1
TON    T38, +5
Network 3
LD     SM0.0
=      L60.0
LD     T37
A      一次抬起:M12.7
A      EMBotton:I0.7
AN     压停PC:M4.0
=      L63.7
LD     L60.0
CALL   AXIS0_GOTO:SBR6, L63.7, 0.0, 10.0, 0, 下压轴停止信号:M13.0, 下压轴done:M8.2, 下压轴错误:VB308, 下压轴pos:VD420, 下压轴速度:VD408
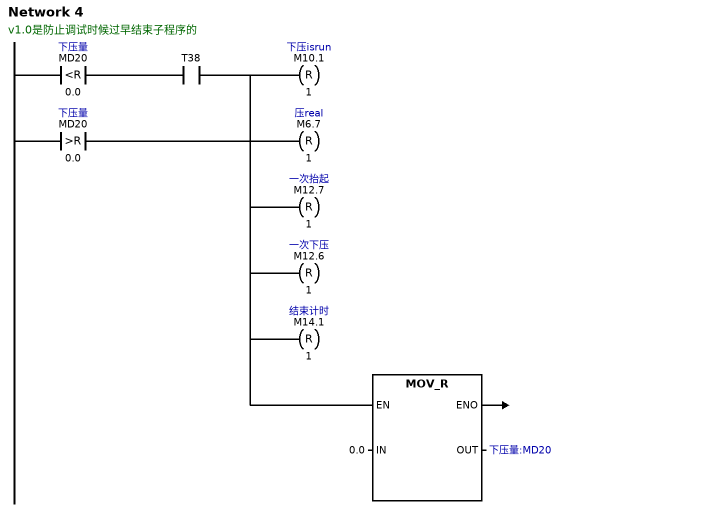
Network 4
// v1.0是防止调试时候过早结束子程序的
LDR<   下压量:MD20, 0.0
A      T38
OR>    下压量:MD20, 0.0
R      下压isrun:M10.1, 1
R      压real:M6.7, 1
R      一次抬起:M12.7, 1
R      一次下压:M12.6, 1
R      结束计时:M14.1, 1
MOVR   0.0, 下压量:MD20
END_SUBROUTINE_BLOCK

// SBR4: protected block, not included

// SBR5: protected block, not included

// SBR6: protected block, not included

// SBR7: protected block, not included

// SBR8: protected block, not included

// SBR9: protected block, not included

// SBR10: protected block, not included

// SBR11: protected block, not included

// SBR12: protected block, not included

// SBR13: protected block, not included

// SBR14: protected block, not included

// SBR15: protected block, not included

// SBR16: protected block, not included

// SBR17: protected block, not included

// SBR18: protected block, not included

// SBR19: protected block, not included

// SBR20: protected block, not included

// SBR21: protected block, not included

// SBR22: protected block, not included

// SBR23: protected block, not included

// SBR24: protected block, not included

// SBR25: protected block, not included

// SBR26: protected block, not included

// SBR27: protected block, not included

// SBR28: protected block, not included

// SBR29: protected block, not included

// SBR30: protected block, not included

// SBR31: protected block, not included

// SBR32: protected block, not included

// SBR33: protected block, not included

SUBROUTINE_BLOCK 通讯:SBR34
TITLE=子程序注释
BEGIN
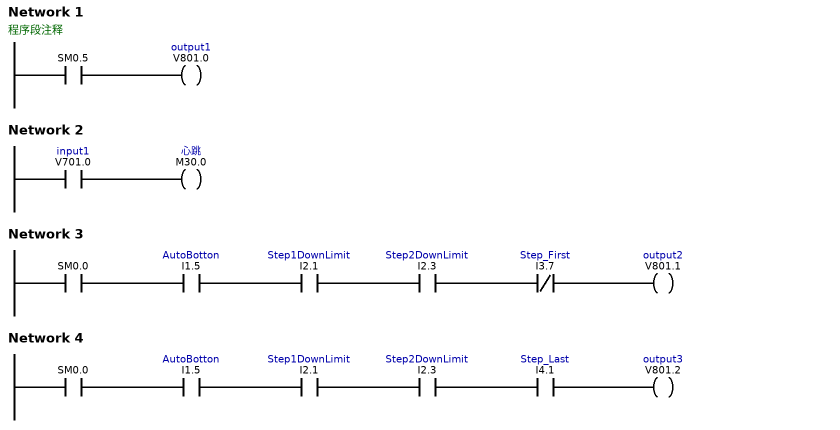
Network 1
// 程序段注释
LD     SM0.5
=      output1:V801.0
Network 2
LD     input1:V701.0
=      心跳:M30.0
Network 3
LD     SM0.0
A      AutoBotton:I1.5
A      Step1DownLimit:I2.1
A      Step2DownLimit:I2.3
AN     Step_First:I3.7
=      output2:V801.1
Network 4
LD     SM0.0
A      AutoBotton:I1.5
A      Step1DownLimit:I2.1
A      Step2DownLimit:I2.3
A      Step_Last:I4.1
=      output3:V801.2
END_SUBROUTINE_BLOCK

SUBROUTINE_BLOCK 夹爪_备压:SBR35
TITLE=子程序注释
BEGIN
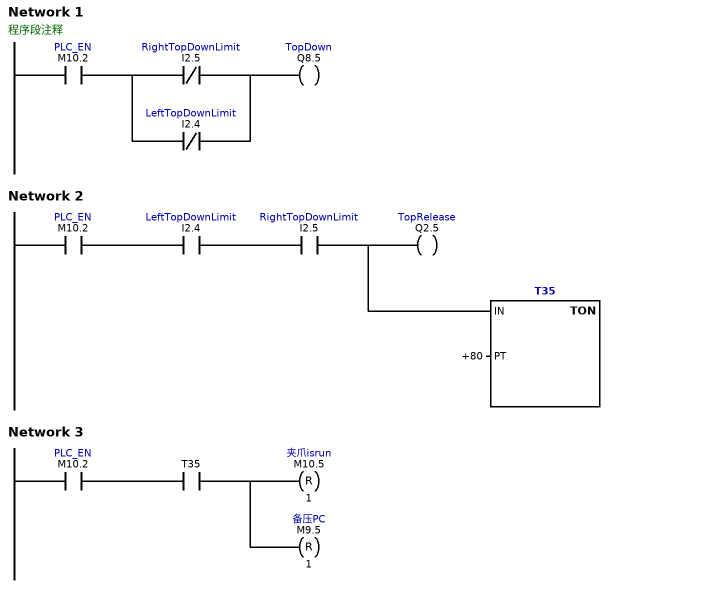
Network 1
// 程序段注释
LD     PLC_EN:M10.2
LDN    RightTopDownLimit:I2.5
ON     LeftTopDownLimit:I2.4
ALD
=      TopDown:Q8.5
Network 2
LD     PLC_EN:M10.2
A      LeftTopDownLimit:I2.4
A      RightTopDownLimit:I2.5
=      TopRelease:Q2.5
TON    T35, +80
Network 3
LD     PLC_EN:M10.2
A      T35
R      夹爪isrun:M10.5, 1
R      备压PC:M9.5, 1
Network 4
// 程序段注释
END_SUBROUTINE_BLOCK
